{attribute 'qualified_only'}
VAR_GLOBAL
	// 1. Axes available for control by EMs
	Axis : ARRAY[1..MAX_AXES] OF FB_Component_BasicAxis;
END_VAR

VAR_GLOBAL CONSTANT
	MAX_AXES : INT := 10;
END_VAR

(* stored: Version 1.1.0.1
   GVL GVL_Axes: Id {629b614c-b48f-44cc-a574-42717181726e} *)
